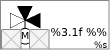
VISUALIZATION StellAntrieb_MB_Valve_AB_Left_RB_CheckEnabled  // 110x50
VAR_INPUT
    ITF_STELLANTRIEB_IN   	:   ITF_STELLANTRIEB;
	stExklParameter			:	STRING[40];
END_VAR
    Frame (0,0 50x50), invisible if: NOT ITF_STELLANTRIEB_IN.proIsEnabled
        shows Icon_MB_AB_L(ITF_STELLANTRIEB_IN := ITF_STELLANTRIEB_IN)
    Frame (50,25 60x25), invisible if: NOT ITF_STELLANTRIEB_IN.proIsEnabled
        shows ValueDwnUp(ITF_STELLANTRIEB_IN := ITF_STELLANTRIEB_IN, uiTextAusrichtung := 4)
    Rectangle (0,0 110x50)
        OnMouseClick:  Dialog=StellAntrieb_POPUP, Parameters={stExklParameter: stExklParameter, ITF_STELLANTRIEBIN: ITF_STELLANTRIEB_IN, uiPopUpGruppe: 0}, OpenCentered=True
END_VISUALIZATION

// 40 Visualizations/ICON/StellAntrieb_RIGHT/Motor_Below/Valve_AB_Right/StellAntrieb_MB_Valve_AB_Right_RB_CheckEnabled
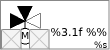
VISUALIZATION StellAntrieb_MB_Valve_AB_Right_RB_CheckEnabled  // 110x50
VAR_INPUT
    ITF_STELLANTRIEB_IN   	:   ITF_STELLANTRIEB;
	stExklParameter			:	STRING[40];
END_VAR
    Frame (0,0 50x50), invisible if: NOT ITF_STELLANTRIEB_IN.proIsEnabled
        shows Icon_MB_AB_R(ITF_STELLANTRIEB_IN := ITF_STELLANTRIEB_IN)
    Frame (50,25 60x25), invisible if: NOT ITF_STELLANTRIEB_IN.proIsEnabled
        shows ValueDwnUp(ITF_STELLANTRIEB_IN := ITF_STELLANTRIEB_IN, uiTextAusrichtung := 4)
    Rectangle (0,0 110x50)
        OnMouseClick:  Dialog=StellAntrieb_POPUP, Parameters={stExklParameter: stExklParameter, ITF_STELLANTRIEBIN: ITF_STELLANTRIEB_IN, uiPopUpGruppe: 0}, OpenCentered=True
END_VISUALIZATION

// 40 Visualizations/ICON/StellAntrieb_RIGHT/Motor_Below/Valve_AB_Left/StellAntrieb_MB_Valve_AB_Left_RB_CheckQuerry
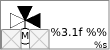
VISUALIZATION StellAntrieb_MB_Valve_AB_Left_RB_CheckQuerry  // 110x50
VAR_INPUT
    ITF_STELLANTRIEB_IN   	:   ITF_STELLANTRIEB;
	stExklParameter			:	STRING[40];
END_VAR
    Frame (0,0 110x50)
        shows StellAntrieb_MB_Valve_AB_Left_RB_CheckEnabled(ITF_STELLANTRIEB_IN := ITF_STELLANTRIEB_IN, stExklParameter := stExklParameter)
END_VISUALIZATION

// 40 Visualizations/ICON/StellAntrieb_RIGHT/Motor_Below/Valve_AB_Left/StellAntrieb_MB_Valve_AB_Left_Txt_R_Below
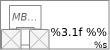
VISUALIZATION StellAntrieb_MB_Valve_AB_Left_Txt_R_Below  // 110x50
VAR_INPUT
    ITF_STELLANTRIEB_IN   	:   ITF_STELLANTRIEB;	
END_VAR
VAR_INPUT CONSTANT
	stExklParameter			:	STRING[40] := '';
END_VAR
VAR CONSTANT
	uiIconNr				: 	UINT := 20;
END_VAR
    Frame (0,0 110x50), invisible if: NOT fcCheckQuerryReturnIcon(_ITF_In := ITF_STELLANTRIEB_IN,_uiIconNr_In := uiIconNr)
        shows StellAntrieb_MB_Valve_AB_Left_RB_CheckQuerry(ITF_STELLANTRIEB_IN := ITF_STELLANTRIEB_IN, stExklParameter := stExklParameter)
        shows Icon()
END_VISUALIZATION

// 40 Visualizations/ICON/StellAntrieb_RIGHT/Motor_Below/Valve_AB_Right/StellAntrieb_MB_Valve_AB_Right_RB_CheckQuerry
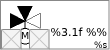
VISUALIZATION StellAntrieb_MB_Valve_AB_Right_RB_CheckQuerry  // 110x50
VAR_INPUT
    ITF_STELLANTRIEB_IN   	:   ITF_STELLANTRIEB;
	stExklParameter			:	STRING[40];
END_VAR
    Frame (0,0 110x50)
        shows StellAntrieb_MB_Valve_AB_Right_RB_CheckEnabled(ITF_STELLANTRIEB_IN := ITF_STELLANTRIEB_IN, stExklParameter := stExklParameter)
END_VISUALIZATION

// 40 Visualizations/ICON/StellAntrieb_RIGHT/Motor_Below/Valve_AB_Right/StellAntrieb_MB_Valve_AB_Right_Txt_R_Below
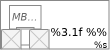
VISUALIZATION StellAntrieb_MB_Valve_AB_Right_Txt_R_Below  // 110x50
VAR_INPUT
    ITF_STELLANTRIEB_IN   	:   ITF_STELLANTRIEB;	
END_VAR
VAR_INPUT CONSTANT
	stExklParameter			:	STRING[40] := '';
END_VAR
VAR CONSTANT
	uiIconNr				: 	UINT := 21;
END_VAR
    Frame (0,0 110x50), invisible if: NOT fcCheckQuerryReturnIcon(_ITF_In := ITF_STELLANTRIEB_IN,_uiIconNr_In := uiIconNr)
        shows StellAntrieb_MB_Valve_AB_Right_RB_CheckQuerry(ITF_STELLANTRIEB_IN := ITF_STELLANTRIEB_IN, stExklParameter := stExklParameter)
        shows Icon()
END_VISUALIZATION

// 40 Visualizations/ICON/StellAntrieb_RIGHT/Motor_Above/Valve_AB_Right/StellAntrieb_MA_Valve_AB_Right_RA_CheckEnabled
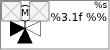
VISUALIZATION StellAntrieb_MA_Valve_AB_Right_RA_CheckEnabled  // 110x50
VAR_INPUT
    ITF_STELLANTRIEB_IN   	:   ITF_STELLANTRIEB;	
	stExklParameter			:	STRING[40];
END_VAR
    Frame (0,0 50x50), invisible if: NOT ITF_STELLANTRIEB_IN.proIsEnabled
        shows Icon_MA_AB_R(ITF_STELLANTRIEB_IN := ITF_STELLANTRIEB_IN)
    Frame (50,0 60x25), invisible if: NOT ITF_STELLANTRIEB_IN.proIsEnabled
        shows ValueUpDwn(ITF_STELLANTRIEB_IN := ITF_STELLANTRIEB_IN, uiTextAusrichtung := 4)
    Rectangle (0,0 110x50)
        OnMouseClick:  Dialog=StellAntrieb_POPUP, Parameters={stExklParameter: stExklParameter, ITF_STELLANTRIEBIN: ITF_STELLANTRIEB_IN, uiPopUpGruppe: 0}, OpenCentered=True
END_VISUALIZATION

// 40 Visualizations/ICON/StellAntrieb_RIGHT/Motor_Above/Valve_AB_Left/StellAntrieb_MA_Valve_AB_Left_RA_CheckEnabled
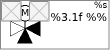
VISUALIZATION StellAntrieb_MA_Valve_AB_Left_RA_CheckEnabled  // 110x50
VAR_INPUT
    ITF_STELLANTRIEB_IN   	:   ITF_STELLANTRIEB;	
	stExklParameter			:	STRING[40];
END_VAR
    Frame (0,0 50x50), invisible if: NOT ITF_STELLANTRIEB_IN.proIsEnabled
        shows Icon_MA_AB_L(ITF_STELLANTRIEB_IN := ITF_STELLANTRIEB_IN)
    Frame (50,0 60x25), invisible if: NOT ITF_STELLANTRIEB_IN.proIsEnabled
        shows ValueUpDwn(ITF_STELLANTRIEB_IN := ITF_STELLANTRIEB_IN, uiTextAusrichtung := 4)
    Rectangle (0,0 110x50)
        OnMouseClick:  Dialog=StellAntrieb_POPUP, Parameters={stExklParameter: stExklParameter, ITF_STELLANTRIEBIN: ITF_STELLANTRIEB_IN, uiPopUpGruppe: 0}, OpenCentered=True
END_VISUALIZATION

// 40 Visualizations/ICON/StellAntrieb_RIGHT/Motor_Above/Valve_AB_Right/StellAntrieb_MA_Valve_AB_Right_RA_CheckQuerry
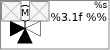
VISUALIZATION StellAntrieb_MA_Valve_AB_Right_RA_CheckQuerry  // 110x50
VAR_INPUT
    ITF_STELLANTRIEB_IN   	:   ITF_STELLANTRIEB;
	stExklParameter			:	STRING[40];
END_VAR
    Frame (0,0 110x50)
        shows StellAntrieb_MA_Valve_AB_Right_RA_CheckEnabled(ITF_STELLANTRIEB_IN := ITF_STELLANTRIEB_IN, stExklParameter := stExklParameter)
END_VISUALIZATION

// 40 Visualizations/ICON/StellAntrieb_RIGHT/Motor_Above/Valve_AB_Right/StellAntrieb_MA_Valve_AB_Right_Txt_R_Above
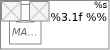
VISUALIZATION StellAntrieb_MA_Valve_AB_Right_Txt_R_Above  // 110x50
VAR_INPUT
    ITF_STELLANTRIEB_IN   	:   ITF_STELLANTRIEB;	
END_VAR
VAR_INPUT CONSTANT
	stExklParameter			:	STRING[40] := '';
END_VAR
VAR CONSTANT
	uiIconNr				: 	UINT := 17;
END_VAR
    Frame (0,0 110x50), invisible if: NOT fcCheckQuerryReturnIcon(_ITF_In := ITF_STELLANTRIEB_IN,_uiIconNr_In := uiIconNr)
        shows StellAntrieb_MA_Valve_AB_Right_RA_CheckQuerry(ITF_STELLANTRIEB_IN := ITF_STELLANTRIEB_IN, stExklParameter := stExklParameter)
        shows Icon()
END_VISUALIZATION

// 40 Visualizations/ICON/StellAntrieb_RIGHT/Motor_Above/Valve_AB_Left/StellAntrieb_MA_Valve_AB_Left_RA_CheckQuerry
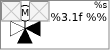
VISUALIZATION StellAntrieb_MA_Valve_AB_Left_RA_CheckQuerry  // 110x50
VAR_INPUT
    ITF_STELLANTRIEB_IN   	:   ITF_STELLANTRIEB;
	stExklParameter			:	STRING[40];
END_VAR
    Frame (0,0 110x50)
        shows StellAntrieb_MA_Valve_AB_Left_RA_CheckEnabled(ITF_STELLANTRIEB_IN := ITF_STELLANTRIEB_IN, stExklParameter := stExklParameter)
END_VISUALIZATION

// 40 Visualizations/ICON/StellAntrieb_RIGHT/Motor_Above/Valve_AB_Left/StellAntrieb_MA_Valve_AB_Left_Txt_R_Above
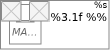
VISUALIZATION StellAntrieb_MA_Valve_AB_Left_Txt_R_Above  // 110x50
VAR_INPUT
    ITF_STELLANTRIEB_IN   	:   ITF_STELLANTRIEB;	
END_VAR
VAR_INPUT CONSTANT
	stExklParameter			:	STRING[40] := '';
END_VAR
VAR CONSTANT
	uiIconNr				: 	UINT := 16;
END_VAR
    Frame (0,0 110x50), invisible if: NOT fcCheckQuerryReturnIcon(_ITF_In := ITF_STELLANTRIEB_IN,_uiIconNr_In := uiIconNr)
        shows StellAntrieb_MA_Valve_AB_Left_RA_CheckQuerry(ITF_STELLANTRIEB_IN := ITF_STELLANTRIEB_IN, stExklParameter := stExklParameter)
        shows Icon()
END_VISUALIZATION

// 40 Visualizations/ICON/StellAntrieb_LEFT/Motor_Below/Valve_AB_Left/StellAntrieb_MB_Valve_AB_Left_LB_CheckEnabled
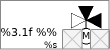
VISUALIZATION StellAntrieb_MB_Valve_AB_Left_LB_CheckEnabled  // 110x50
VAR_INPUT
    ITF_STELLANTRIEB_IN   	:   ITF_STELLANTRIEB;
	stExklParameter			:	STRING[40];
END_VAR
    Frame (61,0 50x50), invisible if: NOT ITF_STELLANTRIEB_IN.proIsEnabled
        shows Icon_MB_AB_L(ITF_STELLANTRIEB_IN := ITF_STELLANTRIEB_IN)
    Frame (0,25 60x25), invisible if: NOT ITF_STELLANTRIEB_IN.proIsEnabled
        shows ValueDwnUp(ITF_STELLANTRIEB_IN := ITF_STELLANTRIEB_IN, uiTextAusrichtung := 6)
    Rectangle (0,0 110x50)
        OnMouseClick:  Dialog=StellAntrieb_POPUP, Parameters={stExklParameter: stExklParameter, ITF_STELLANTRIEBIN: ITF_STELLANTRIEB_IN, uiPopUpGruppe: 0}, OpenCentered=True
END_VISUALIZATION

// 40 Visualizations/ICON/StellAntrieb_RIGHT/Motor_Right/Valve_AB_Up/Above/StellAntrieb_MR_Valve_AB_Up_RA_CheckEnabled
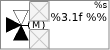
VISUALIZATION StellAntrieb_MR_Valve_AB_Up_RA_CheckEnabled  // 110x50
VAR_INPUT
    ITF_STELLANTRIEB_IN   	:   ITF_STELLANTRIEB;	
	stExklParameter			:	STRING[40];
END_VAR
    Frame (0,0 50x50), invisible if: NOT ITF_STELLANTRIEB_IN.proIsEnabled
        shows Icon_MR_AB_Up(ITF_STELLANTRIEB_IN := ITF_STELLANTRIEB_IN)
    Frame (50,0 60x25), invisible if: NOT ITF_STELLANTRIEB_IN.proIsEnabled
        shows ValueUpDwn(ITF_STELLANTRIEB_IN := ITF_STELLANTRIEB_IN, uiTextAusrichtung := 4)
    Rectangle (0,0 110x50)
        OnMouseClick:  Dialog=StellAntrieb_POPUP, Parameters={stExklParameter: stExklParameter, ITF_STELLANTRIEBIN: ITF_STELLANTRIEB_IN, uiPopUpGruppe: 0}, OpenCentered=True
END_VISUALIZATION

// 40 Visualizations/ICON/StellAntrieb_RIGHT/Motor_Right/Valve_AB_Up/Above/StellAntrieb_MR_Valve_AB_Up_RA_CheckQuerry
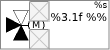
VISUALIZATION StellAntrieb_MR_Valve_AB_Up_RA_CheckQuerry  // 110x50
VAR_INPUT
    ITF_STELLANTRIEB_IN   	:   ITF_STELLANTRIEB;	
	stExklParameter			:	STRING[40];
END_VAR
    Frame (0,0 110x50)
        shows StellAntrieb_MR_Valve_AB_Up_RA_CheckEnabled(ITF_STELLANTRIEB_IN := ITF_STELLANTRIEB_IN, stExklParameter := stExklParameter)
END_VISUALIZATION

// 40 Visualizations/ICON/StellAntrieb_LEFT/Motor_Below/Valve_AB_Left/StellAntrieb_MB_Valve_AB_Left_LB_CheckQuerry
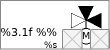
VISUALIZATION StellAntrieb_MB_Valve_AB_Left_LB_CheckQuerry  // 110x50
VAR_INPUT
    ITF_STELLANTRIEB_IN   	:   ITF_STELLANTRIEB;
	stExklParameter			:	STRING[40];
END_VAR
    Frame (0,0 110x50)
        shows StellAntrieb_MB_Valve_AB_Left_LB_CheckEnabled(ITF_STELLANTRIEB_IN := ITF_STELLANTRIEB_IN, stExklParameter := stExklParameter)
END_VISUALIZATION

// 40 Visualizations/ICON/StellAntrieb_LEFT/Motor_Below/Valve_AB_Left/StellAntrieb_MB_Valve_AB_Left_Txt_L_Below
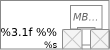
VISUALIZATION StellAntrieb_MB_Valve_AB_Left_Txt_L_Below  // 110x50
VAR_INPUT
    ITF_STELLANTRIEB_IN   	:   ITF_STELLANTRIEB;	
END_VAR
VAR_INPUT CONSTANT
	stExklParameter			:	STRING[40] := '';
END_VAR
VAR CONSTANT
	uiIconNr				: 	UINT := 4;
END_VAR
    Frame (0,0 110x50), invisible if: NOT fcCheckQuerryReturnIcon(_ITF_In := ITF_STELLANTRIEB_IN,_uiIconNr_In := uiIconNr)
        shows StellAntrieb_MB_Valve_AB_Left_LB_CheckQuerry(ITF_STELLANTRIEB_IN := ITF_STELLANTRIEB_IN, stExklParameter := stExklParameter)
        shows Icon()
END_VISUALIZATION

// 40 Visualizations/ICON/StellAntrieb_LEFT/Motor_Below/Valve_AB_Right/StellAntrieb_MB_Valve_AB_Right_LB_CheckEnabled
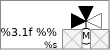
VISUALIZATION StellAntrieb_MB_Valve_AB_Right_LB_CheckEnabled  // 110x50
VAR_INPUT
    ITF_STELLANTRIEB_IN   	:   ITF_STELLANTRIEB;
	stExklParameter			:	STRING[40];
END_VAR
    Frame (61,0 50x50), invisible if: NOT ITF_STELLANTRIEB_IN.proIsEnabled
        shows Icon_MB_AB_R(ITF_STELLANTRIEB_IN := ITF_STELLANTRIEB_IN)
    Frame (0,25 60x25), invisible if: NOT ITF_STELLANTRIEB_IN.proIsEnabled
        shows ValueDwnUp(ITF_STELLANTRIEB_IN := ITF_STELLANTRIEB_IN, uiTextAusrichtung := 6)
    Rectangle (0,0 110x50)
        OnMouseClick:  Dialog=StellAntrieb_POPUP, Parameters={stExklParameter: stExklParameter, ITF_STELLANTRIEBIN: ITF_STELLANTRIEB_IN, uiPopUpGruppe: 0}, OpenCentered=True
END_VISUALIZATION

// 40 Visualizations/ICON/StellAntrieb_LEFT/Motor_Above/Valve_AB_Left/StellAntrieb_MA_Valve_AB_Left_LA_CheckEnabled
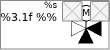
VISUALIZATION StellAntrieb_MA_Valve_AB_Left_LA_CheckEnabled  // 110x50
VAR_INPUT
    ITF_STELLANTRIEB_IN   :   ITF_STELLANTRIEB;
	stExklParameter		:	STRING[40];
END_VAR
    Frame (61,0 50x50), invisible if: NOT ITF_STELLANTRIEB_IN.proIsEnabled
        shows Icon_MA_AB_L(ITF_STELLANTRIEB_IN := ITF_STELLANTRIEB_IN)
    Frame (0,0 60x25), invisible if: NOT ITF_STELLANTRIEB_IN.proIsEnabled
        shows ValueUpDwn(ITF_STELLANTRIEB_IN := ITF_STELLANTRIEB_IN, uiTextAusrichtung := 6)
    Rectangle (0,0 110x50)
        OnMouseClick:  Dialog=StellAntrieb_POPUP, Parameters={stExklParameter: stExklParameter, ITF_STELLANTRIEBIN: ITF_STELLANTRIEB_IN, uiPopUpGruppe: 0}, OpenCentered=True
END_VISUALIZATION

// 40 Visualizations/ICON/StellAntrieb_RIGHT/Motor_Right/Valve_AB_Up/Above/StellAntrieb_MR_Valve_AB_Up_Txt_R_Above
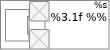
VISUALIZATION StellAntrieb_MR_Valve_AB_Up_Txt_R_Above  // 110x50
VAR_INPUT
    ITF_STELLANTRIEB_IN   	:   ITF_STELLANTRIEB;	
END_VAR
VAR_INPUT CONSTANT
	stExklParameter			:	STRING[40] := '';
END_VAR
VAR CONSTANT
	uiIconNr				: 	UINT := 26;
END_VAR
    Frame (0,0 110x50), invisible if: NOT fcCheckQuerryReturnIcon(_ITF_In := ITF_STELLANTRIEB_IN,_uiIconNr_In := uiIconNr)
        shows StellAntrieb_MR_Valve_AB_Up_RA_CheckQuerry(ITF_STELLANTRIEB_IN := ITF_STELLANTRIEB_IN, stExklParameter := stExklParameter)
        shows Icon()
END_VISUALIZATION

// 40 Visualizations/ICON/StellAntrieb_LEFT/Motor_Above/Valve_AB_Left/StellAntrieb_MA_Valve_AB_Left_LA_CheckQuerry
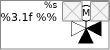
VISUALIZATION StellAntrieb_MA_Valve_AB_Left_LA_CheckQuerry  // 110x50
VAR_INPUT
    ITF_STELLANTRIEB_IN   	:   ITF_STELLANTRIEB;
	stExklParameter			:	STRING[40];
END_VAR
    Frame (0,0 110x50)
        shows StellAntrieb_MA_Valve_AB_Left_LA_CheckEnabled(ITF_STELLANTRIEB_IN := ITF_STELLANTRIEB_IN, stExklParameter := stExklParameter)
END_VISUALIZATION

// 40 Visualizations/ICON/StellAntrieb_LEFT/Motor_Above/Valve_AB_Left/StellAntrieb_MA_Valve_AB_Left_Txt_L_Above
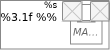
VISUALIZATION StellAntrieb_MA_Valve_AB_Left_Txt_L_Above  // 110x50
VAR_INPUT
    ITF_STELLANTRIEB_IN   	:   ITF_STELLANTRIEB;	
END_VAR
VAR_INPUT CONSTANT
	stExklParameter			:	STRING[40] := '';
END_VAR
VAR CONSTANT
	uiIconNr				: UINT := 0;
END_VAR
    Frame (0,0 110x50), invisible if: NOT fcCheckQuerryReturnIcon(_ITF_In := ITF_STELLANTRIEB_IN,_uiIconNr_In := uiIconNr)
        shows StellAntrieb_MA_Valve_AB_Left_LA_CheckQuerry(ITF_STELLANTRIEB_IN := ITF_STELLANTRIEB_IN, stExklParameter := stExklParameter)
        shows Icon()
END_VISUALIZATION

// 40 Visualizations/ICON/StellAntrieb_LEFT/Motor_Above/Valve_AB_Right/StellAntrieb_MA_Valve_AB_Right_LA_CheckEnabled
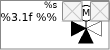
VISUALIZATION StellAntrieb_MA_Valve_AB_Right_LA_CheckEnabled  // 110x50
VAR_INPUT
    ITF_STELLANTRIEB_IN   	:   ITF_STELLANTRIEB;
	stExklParameter			:	STRING[40];
END_VAR
    Frame (61,0 50x50), invisible if: NOT ITF_STELLANTRIEB_IN.proIsEnabled
        shows Icon_MA_AB_R(ITF_STELLANTRIEB_IN := ITF_STELLANTRIEB_IN)
    Frame (0,0 60x25), invisible if: NOT ITF_STELLANTRIEB_IN.proIsEnabled
        shows ValueUpDwn(ITF_STELLANTRIEB_IN := ITF_STELLANTRIEB_IN, uiTextAusrichtung := 6)
    Rectangle (0,0 110x50)
        OnMouseClick:  Dialog=StellAntrieb_POPUP, Parameters={stExklParameter: stExklParameter, ITF_STELLANTRIEBIN: ITF_STELLANTRIEB_IN, uiPopUpGruppe: 0}, OpenCentered=True
END_VISUALIZATION

// 40 Visualizations/ICON/StellAntrieb_RIGHT/Motor_Right/Valve_AB_Up/Below/StellAntrieb_MR_Valve_AB_Up_RB_CheckEnabled
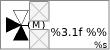
VISUALIZATION StellAntrieb_MR_Valve_AB_Up_RB_CheckEnabled  // 110x50
VAR_INPUT
    ITF_STELLANTRIEB_IN   	:   ITF_STELLANTRIEB;
	stExklParameter			:	STRING[40];
END_VAR
    Frame (0,0 50x50), invisible if: NOT ITF_STELLANTRIEB_IN.proIsEnabled
        shows Icon_MR_AB_Up(ITF_STELLANTRIEB_IN := ITF_STELLANTRIEB_IN)
    Frame (50,25 60x25), invisible if: NOT ITF_STELLANTRIEB_IN.proIsEnabled
        shows ValueDwnUp(ITF_STELLANTRIEB_IN := ITF_STELLANTRIEB_IN, uiTextAusrichtung := 4)
    Rectangle (0,0 110x50)
        OnMouseClick:  Dialog=StellAntrieb_POPUP, Parameters={stExklParameter: stExklParameter, ITF_STELLANTRIEBIN: ITF_STELLANTRIEB_IN, uiPopUpGruppe: 0}, OpenCentered=True
END_VISUALIZATION

// 40 Visualizations/ICON/StellAntrieb_RIGHT/Motor_Right/Valve_AB_Up/Below/StellAntrieb_MR_Valve_AB_Up_RB_CheckQuerry
